FUNCTION_BLOCK Test_TStreamBufferResizes EXTENDS T_UnitTestBase
VAR
    Stream : T_Stream(StreamLength := 2);
END_VAR

METHOD  Init
VAR_INPUT
END_VAR
END_METHOD

{attribute 'analysis' := '-33'} // inhibit unused variable warning
METHOD RunTest
Stream.Init(2);

Stream.Add_INT(1234);
Stream.Add_INT(1235);
Stream.Add_INT(1236);
Stream.Add_INT(1237);

AssertEquals_UDINT(Expected     := 8,
                   Actual       := Stream.WritePosition,
                   Message := 'Stream.WritePosition');

AssertEquals_UDINT(Expected     := 8,
                   Actual       := Stream.StreamLength,
                   Message := 'Stream.StreamLength');

Stream.SetReadPosition(0);

AssertEquals_INT(Expected     := 1234,
                 Actual       := Stream.Read_INT(),
                 Message := 'Stream.ReadInt()');

AssertEquals_UDINT(Expected     := 2,
                   Actual       := Stream.ReadPosition,
                   Message := 'Stream.ReadPosition');

TestCompleted := TRUE;
END_METHOD

END_FUNCTION_BLOCK

(* stored: Version 1.1.0.1, ProductVersion 3.1.4024.12
   POU Test_TStreamBufferResizes: Id {1a895df7-9bb9-473c-8f5b-b5602d113553}, SpecialFunc None
   Method Init: Id {6abb7507-a7c1-40ce-a817-9da9503c0055}
   Method RunTest: Id {5b3bad08-85d4-4d68-892f-45ee54a63213} *)
